INTERFACE I_PersistantEventStorage

METHOD StoreEvent : BOOL
VAR_INPUT
	stEvent : ST_Event;
END_VAR
END_METHOD

END_INTERFACE

(* stored: Version 1.1.0.1, ProductVersion 3.1.4024.12
   Itf I_PersistantEventStorage: Id {347bcdf8-730c-42c3-92df-4c8eca5a3b12}
   Method StoreEvent: Id {ddf4ec10-a567-466a-aecd-65637427ca13} *)
